FUNCTION alg_M_Distributing_a_Dresetled : BOOL
VAR_INPUT
	state: STATE;
END_VAR

alg_M_Distributing_a_Dresetled := ((((((((state.dvar_M_Distributing) <> (elit_wait_start)) AND ((state.dvar_M_Distributing) <> (elit_init2))) AND ((state.dvar_M_Distributing) <> (elit_droppoint))) AND ((state.dvar_M_Distributing) <> (elit_movetopickup))) AND ((state.dvar_M_Distributing) <> (elit_down))) AND ((state.dvar_M_Distributing) <> (elit_gopickup))) AND ((state.dvar_M_Distributing) <> (elit_goback))) AND ((state.dvar_M_Distributing) <> (elit_stop));

END_FUNCTION

(* stored: Version 1.1.0.1, ProductVersion 3.1.4022.18
   POU alg_M_Distributing_a_Dresetled: Id {0dac78ee-a8eb-4b54-b2fe-97f7fdc4b34c}, SpecialFunc None *)
